FUNCTION_BLOCK FB_Extrution
VAR_INPUT
	bEnable : BOOL;
	bStart : BOOL;
	bReset : BOOL;
	bEstop : BOOL;
	lrExtrudtionDistance : LREAL;
	lrFeedRate : LREAL;
END_VAR
VAR_OUTPUT
	bHotendEnable: BOOL;
	lrHotendTemp: LREAL;
	bExtrusionDone : BOOL;
END_VAR
VAR
	fbHotEndTempControl : FB_TempControl;
	iStep : INT :=0;
END_VAR

CASE iStep OF
0: (* Idle *)
	IF bEnable THEN
		iStep :=10;
	END_IF
10: (* Start Heating *)
	
	fbHotEndTempControl(
			bEnabled:= bEnable, 
			lrPV:= , 
			lrSP:= , 
			iOutput=> , 
			bError=> , 
			eErrorId=> );

END_CASE

END_FUNCTION_BLOCK

(* stored: Version 1.1.0.1, ProductVersion 3.1.4024.2
   POU FB_Extrution: Id {7c001826-9b88-46ee-bbcb-f265d4fe38e4}, SpecialFunc None *)
